// TIA Portal V17 export
// export: Created 2025-03-10T12:18:27.772084Z, ExportSetting WithDefaults, DisplayName Totally Integrated Automation Portal, DisplayVersion V17 Update 8, DisplayName TIA Portal Openness, DisplayVersion V17 Update 8, DisplayName TIA Portal Version Control Interface, DisplayVersion V17, DisplayName SINAMICS Startdrive Advanced, DisplayVersion V17 SP2, DisplayName SINAMICS Startdrive G110M, G120, G120C, G120D, G120P, G115D, DisplayVersion V17 SP2, DisplayName SINAMICS Startdrive G130, G150, S120, S150, SINAMICS MV, S210, DisplayVersion V17 SP2, DisplayName STEP 7 Professional, DisplayVersion V17 Update 8, DisplayName SINUMERIK ONE STEP 7 Toolbox, DisplayVersion V17 Update 12, DisplayName SINUMERIK 840D sl STEP 7 Toolbox, DisplayVersion V17 Update 12, DisplayName STEP 7 Safety, DisplayVersion V17 Update 6, DisplayName WinCC Advanced, DisplayVersion V17 Update 8
FUNCTION "FC2000_MACHINE_MODES" : Void   // FC2000, LAD
{ S7_Optimized_Access := 'FALSE' }
AUTHOR : ETXETAR
VERSION : 1.0
// stored: AutoNumber false, IsIECCheckEnabled false, SetENOAutomatically false, UDAEnableTagReadback false
BEGIN

REGION Network 1: OPTIONS OFF
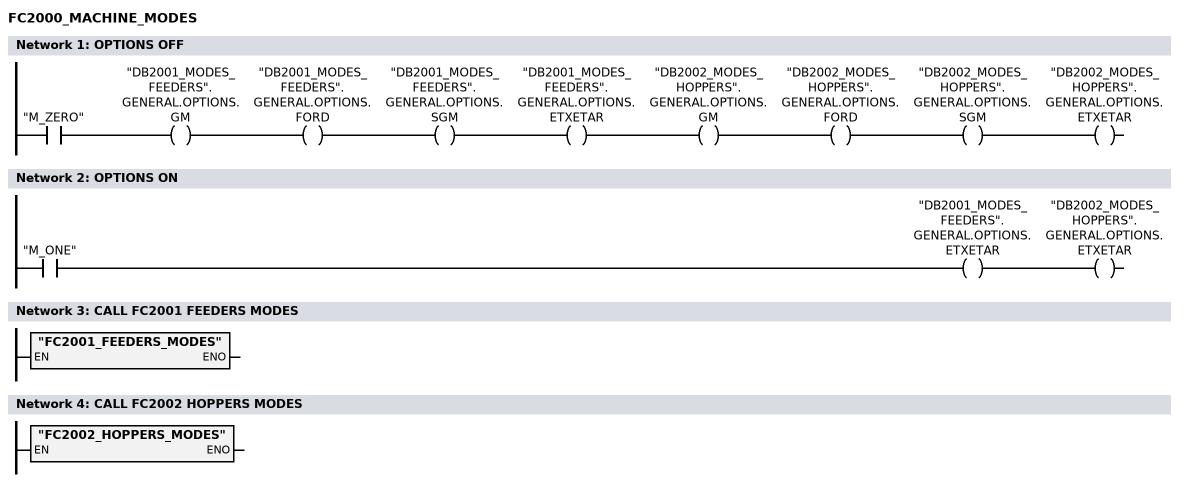
   RUNG wire#powerrail
      Contact( "M_ZERO" )
      Coil( "DB2001_MODES_FEEDERS".GENERAL.OPTIONS.GM )
      Coil( "DB2001_MODES_FEEDERS".GENERAL.OPTIONS.FORD )
      Coil( "DB2001_MODES_FEEDERS".GENERAL.OPTIONS.SGM )
      Coil( "DB2001_MODES_FEEDERS".GENERAL.OPTIONS.ETXETAR )
      Coil( "DB2002_MODES_HOPPERS".GENERAL.OPTIONS.GM )
      Coil( "DB2002_MODES_HOPPERS".GENERAL.OPTIONS.FORD )
      Coil( "DB2002_MODES_HOPPERS".GENERAL.OPTIONS.SGM )
      Coil( "DB2002_MODES_HOPPERS".GENERAL.OPTIONS.ETXETAR )
   END_RUNG
   // the same network as SCL:
   "DB2001_MODES_FEEDERS".GENERAL.OPTIONS.GM := "M_ZERO";
   "DB2001_MODES_FEEDERS".GENERAL.OPTIONS.FORD := "M_ZERO";
   "DB2001_MODES_FEEDERS".GENERAL.OPTIONS.SGM := "M_ZERO";
   "DB2001_MODES_FEEDERS".GENERAL.OPTIONS.ETXETAR := "M_ZERO";
   "DB2002_MODES_HOPPERS".GENERAL.OPTIONS.GM := "M_ZERO";
   "DB2002_MODES_HOPPERS".GENERAL.OPTIONS.FORD := "M_ZERO";
   "DB2002_MODES_HOPPERS".GENERAL.OPTIONS.SGM := "M_ZERO";
   "DB2002_MODES_HOPPERS".GENERAL.OPTIONS.ETXETAR := "M_ZERO";
END_REGION

REGION Network 2: OPTIONS ON
   RUNG wire#powerrail
      Contact( "M_ONE" )
      Coil( "DB2001_MODES_FEEDERS".GENERAL.OPTIONS.ETXETAR )
      Coil( "DB2002_MODES_HOPPERS".GENERAL.OPTIONS.ETXETAR )
   END_RUNG
   // the same network as SCL:
   "DB2001_MODES_FEEDERS".GENERAL.OPTIONS.ETXETAR := "M_ONE";
   "DB2002_MODES_HOPPERS".GENERAL.OPTIONS.ETXETAR := "M_ONE";
END_REGION

REGION Network 3: CALL FC2001 FEEDERS MODES
   RUNG wire#powerrail
      "FC2001_FEEDERS_MODES"()
   END_RUNG
   // the same network as SCL:
   "FC2001_FEEDERS_MODES"();
END_REGION

REGION Network 4: CALL FC2002 HOPPERS MODES
   RUNG wire#powerrail
      "FC2002_HOPPERS_MODES"()
   END_RUNG
   // the same network as SCL:
   "FC2002_HOPPERS_MODES"();
END_REGION
END_FUNCTION
